// TIA Portal V18 export
TYPE "AI"
// stored: IsFailsafeCompliant false
   STRUCT
      "FLOW METER" : Int;
      "CONDUCTIVITY METER" : Int;
      "SPARE AI1" : Int;
      "SPARE AI2" : Int;
   END_STRUCT;
END_TYPE
